{attribute 'GeneratedUsingTerminal: EL9550--0000'}
{attribute addProperty BoxType "EL9550--0000"}
{attribute addProperty Description "EL9550 Surge/Overvoltagefilter (Power and system supply)"}
{attribute addProperty Physics "KK"}
{attribute addProperty Id "EL9550"}
{attribute addProperty CRC "2432835511"}
{attribute addProperty Size "0"}
TYPE EL9550_91021FB7 EXTENDS EtcSlaveTerminalBase_947E5A46 :
STRUCT
END_STRUCT
END_TYPE

(* stored: Version 1.2.0.0, ProductVersion 3.1.4024.11
   DUT EL9550_91021FB7: Id {d61ff0e1-2b06-4e86-9625-bcc0b03da352} *)
